{attribute 'hide_all_locals'}
FUNCTION_BLOCK EnableGroup IMPLEMENTS ITask
VAR_INPUT
END_VAR
VAR_OUTPUT
END_VAR
VAR
	groupEnable			: MC_GroupEnable;
	_caGroup			: REFERENCE TO AXES_GROUP_REF;
	State: INT;
	_enableGroup : BOOL;
	_busy : BOOL;
	_error : BOOL;
	_done : BOOL;
END_VAR

CASE State OF
	0:
		IF _enableGroup THEN
			_done := FALSE;
			_error := FALSE;
			_busy := TRUE;
			groupEnable.Execute := TRUE;
			IF groupEnable.Busy THEN
				State := 10;
				_enableGroup := FALSE;
			END_IF
		END_IF
	
	10:
		IF NOT groupEnable.Busy THEN
			IF groupEnable.Done THEN
				_done := TRUE;
			ELSIF groupEnable.Error THEN
				_error := TRUE;
			END_IF
			_busy := FALSE;
			groupEnable.Execute := false;
			State := 0;
		END_IF
END_CASE


groupEnable(AxesGroup := _caGroup);

METHOD Abort : BOOL
groupEnable.Execute := FALSE;
Abort := TRUE;
State := 0;
END_METHOD

PROPERTY Busy : BOOL
GET
Busy := _busy;
END_GET
END_PROPERTY

PROPERTY Done : BOOL
GET
Done := _done;
END_GET
END_PROPERTY

PROPERTY Error : BOOL
GET
Error := _error;
END_GET
END_PROPERTY

METHOD Execute : BOOL
Execute := _enableGroup := true;
END_METHOD

METHOD FB_init : BOOL
VAR_INPUT
	bInitRetains : BOOL; // if TRUE, the retain variables are initialized (warm start / cold start)
	bInCopyCode : BOOL;  // if TRUE, the instance afterwards gets moved into the copy code (online change)
	CAGroup : Reference TO AXES_GROUP_REF;	
END_VAR
_caGroup REF= CAGroup;
END_METHOD

END_FUNCTION_BLOCK

(* stored: Version 1.1.0.1, ProductVersion 3.1.4024.6
   POU EnableGroup: Id {4aa69e18-750b-47d6-bedb-2553dc5fab79}, SpecialFunc None
   Method Abort: Id {17e04b01-8656-466e-9c23-4ab8d0f72204}
   Property Busy: Id {364c0496-b7cf-4336-92c5-3d8e42d78be4}
   Get Get: Id {2ef95a9b-3b3f-4097-b153-f35964b6f7b8}
   Property Done: Id {d75d00ee-cb88-402a-b7d4-68d7ea7d86db}
   Get Get: Id {acafffc2-8692-4c9f-b143-e99b2058dd69}
   Property Error: Id {cd86fecf-4f88-4303-91a8-489d08794c41}
   Get Get: Id {d6a84586-3449-4f32-a83a-5ae32a1e0610}
   Method Execute: Id {6a5805b9-5a55-452f-9758-47e449eaaf6c}
   Method FB_init: Id {0af1d71d-ce8d-4fcd-b1a8-0172895ab235} *)
